FUNCTION_BLOCK PUBLIC FB_Lamp
VAR_OUTPUT
	byLevel			: BYTE;
END_VAR

PROPERTY PUBLIC Level : BYTE
GET
Level := byLevel;
END_GET
END_PROPERTY

METHOD PUBLIC SetLevel : BOOL
VAR_INPUT
	byNewLevel			:	BYTE;
END_VAR
byLevel := byNewLevel;
END_METHOD

END_FUNCTION_BLOCK

(* stored: Version 1.1.0.1, ProductVersion 3.1.4024.12
   POU FB_Lamp: Id {3bca07a4-e6a3-4993-b3ce-cd6208715083}, SpecialFunc None
   Property Level: Id {fd1f9381-9278-4795-8ca0-574ae82e0344}
   Get Get: Id {6bc0711d-44fd-4f5c-aea2-929d8fcabe0d}
   Method SetLevel: Id {ee841ca3-75a6-4352-8c3c-7b2091f6571b} *)
